PROGRAM P_RoomController_Test_CFC
VAR
	fbRoomController	:	FB_RoomController;
	fbmyLight			:	FB_MyLight1;
	fbDelayedLight		:	FB_DelayedLight;
	fbDimmingLight		:	FB_DimmingLight;
	bAllOn				:	BOOL;
	bAllOff				:	BOOL;
	bAllCallMinLevel	:	BOOL;
	aControlLevel		:	ARRAY [1..3] OF BOOL;
	aDimmLevel			:	ARRAY [1..3] OF BYTE;
END_VAR

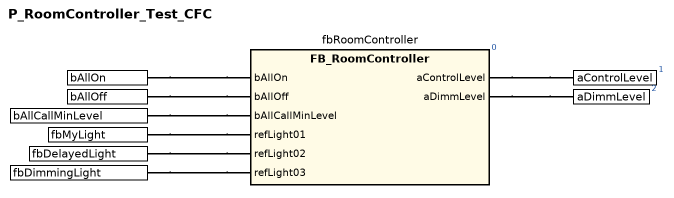
fbRoomController(
    bAllOn := bAllOn,
    bAllOff := bAllOff,
    bAllCallMinLevel := bAllCallMinLevel,
    refLight01 := fbMyLight,
    refLight02 := fbDelayedLight,
    refLight03 := fbDimmingLight); // FB_RoomController
aControlLevel := fbRoomController.aControlLevel;
aDimmLevel := fbRoomController.aDimmLevel;

END_PROGRAM

(* stored: Version 1.1.0.1, ProductVersion 3.1.4024.12
   POU P_RoomController_Test_CFC: Id {a6307abe-a1f8-4cf1-85d9-96120581b71f}, SpecialFunc None *)
